	X =  157.000  mm,	Y =  130.000  mm,	Z =   -1.000 mm,
	W =-180.000 deg,	P =   0.000 deg,	R =    90.000 deg
};
P[6603]{
   GP1:
	UF : 1, UT : 3,		CONFIG : 'N U T, 0, 0, 0',
	X =  157.000  mm,	Y =  130.000  mm,	Z =   15.000 mm,
	W =-180.000 deg,	P =   0.000 deg,	R =    90.000 deg
};
P[6745]{
   GP1:
	UF : 1, UT : 3,		CONFIG : 'N U T, 0, 0, 0',
	X =  34.000  mm,	Y =  136.000  mm,	Z =   15.000 mm,
	W =-180.000 deg,	P =   0.000 deg,	R =    90.000 deg
};
P[6746]{
   GP1:
	UF : 1, UT : 3,		CONFIG : 'N U T, 0, 0, 0',
	X =  34.000  mm,	Y =  136.000  mm,	Z =   -1.000 mm,
	W =-180.000 deg,	P =   0.000 deg,	R =    90.000 deg
};
P[6747]{
   GP1:
	UF : 1, UT : 3,		CONFIG : 'N U T, 0, 0, 0',
	X =  34.000  mm,	Y =  136.000  mm,	Z =   15.000 mm,
	W =-180.000 deg,	P =   0.000 deg,	R =    90.000 deg
};
P[6778]{
   GP1:
	UF : 1, UT : 3,		CONFIG : 'N U T, 0, 0, 0',
	X =  106.000  mm,	Y =  136.000  mm,	Z =   15.000 mm,
	W =-180.000 deg,	P =   0.000 deg,	R =    90.000 deg
};
P[6779]{
   GP1:
	UF : 1, UT : 3,		CONFIG : 'N U T, 0, 0, 0',
	X =  106.000  mm,	Y =  136.000  mm,	Z =   -1.000 mm,
	W =-180.000 deg,	P =   0.000 deg,	R =    90.000 deg
};
P[6780]{
   GP1:
	UF : 1, UT : 3,		CONFIG : 'N U T, 0, 0, 0',
	X =  106.000  mm,	Y =  136.000  mm,	Z =   15.000 mm,
	W =-180.000 deg,	P =   0.000 deg,	R =    90.000 deg
};
P[6988]{
   GP1:
	UF : 1, UT : 3,		CONFIG : 'N U T, 0, 0, 0',
	X =  94.000  mm,	Y =  142.000  mm,	Z =   15.000 mm,
	W =-180.000 deg,	P =   0.000 deg,	R =    90.000 deg
};
P[6989]{
   GP1:
	UF : 1, UT : 3,		CONFIG : 'N U T, 0, 0, 0',
	X =  94.000  mm,	Y =  142.000  mm,	Z =   -1.000 mm,
	W =-180.000 deg,	P =   0.000 deg,	R =    90.000 deg
};
P[6990]{
   GP1:
	UF : 1, UT : 3,		CONFIG : 'N U T, 0, 0, 0',
	X =  94.000  mm,	Y =  142.000  mm,	Z =   15.000 mm,
	W =-180.000 deg,	P =   0.000 deg,	R =    90.000 deg
};
P[7054]{
   GP1:
	UF : 1, UT : 3,		CONFIG : 'N U T, 0, 0, 0',
	X =  22.000  mm,	Y =  145.000  mm,	Z =   15.000 mm,
	W =-180.000 deg,	P =   0.000 deg,	R =    90.000 deg
};
P[7055]{
   GP1:
	UF : 1, UT : 3,		CONFIG : 'N U T, 0, 0, 0',
	X =  22.000  mm,	Y =  145.000  mm,	Z =   -1.000 mm,
	W =-180.000 deg,	P =   0.000 deg,	R =    90.000 deg
};
P[7056]{
   GP1:
	UF : 1, UT : 3,		CONFIG : 'N U T, 0, 0, 0',
	X =  22.000  mm,	Y =  145.000  mm,	Z =   15.000 mm,
	W =-180.000 deg,	P =   0.000 deg,	R =    90.000 deg
};
P[7312]{
   GP1:
	UF : 1, UT : 3,		CONFIG : 'N U T, 0, 0, 0',
	X =  109.000  mm,	Y =  151.000  mm,	Z =   15.000 mm,
	W =-180.000 deg,	P =   0.000 deg,	R =    90.000 deg
};
P[7313]{
   GP1:
	UF : 1, UT : 3,		CONFIG : 'N U T, 0, 0, 0',
	X =  109.000  mm,	Y =  151.000  mm,	Z =   -1.000 mm,
	W =-180.000 deg,	P =   0.000 deg,	R =    90.000 deg
};
P[7314]{
   GP1:
	UF : 1, UT : 3,		CONFIG : 'N U T, 0, 0, 0',
	X =  109.000  mm,	Y =  151.000  mm,	Z =   15.000 mm,
	W =-180.000 deg,	P =   0.000 deg,	R =    90.000 deg
};
P[7414]{
   GP1:
	UF : 1, UT : 3,		CONFIG : 'N U T, 0, 0, 0',
	X =  67.000  mm,	Y =  154.000  mm,	Z =   15.000 mm,
	W =-180.000 deg,	P =   0.000 deg,	R =    90.000 deg
};
P[7415]{
   GP1:
	UF : 1, UT : 3,		CONFIG : 'N U T, 0, 0, 0',
	X =  67.000  mm,	Y =  154.000  mm,	Z =   -1.000 mm,
	W =-180.000 deg,	P =   0.000 deg,	R =    90.000 deg
};
P[7416]{
   GP1:
	UF : 1, UT : 3,		CONFIG : 'N U T, 0, 0, 0',
	X =  67.000  mm,	Y =  154.000  mm,	Z =   15.000 mm,
	W =-180.000 deg,	P =   0.000 deg,	R =    90.000 deg
};
P[7657]{
   GP1:
	UF : 1, UT : 3,		CONFIG : 'N U T, 0, 0, 0',
	X =  151.000  mm,	Y =  160.000  mm,	Z =   15.000 mm,
	W =-180.000 deg,	P =   0.000 deg,	R =    90.000 deg
};
P[7658]{
   GP1:
	UF : 1, UT : 3,		CONFIG : 'N U T, 0, 0, 0',
	X =  151.000  mm,	Y =  160.000  mm,	Z =   -1.000 mm,
	W =-180.000 deg,	P =   0.000 deg,	R =    90.000 deg
};
P[7659]{
   GP1:
	UF : 1, UT : 3,		CONFIG : 'N U T, 0, 0, 0',
	X =  151.000  mm,	Y =  160.000  mm,	Z =   15.000 mm,
	W =-180.000 deg,	P =   0.000 deg,	R =    90.000 deg
};
P[7660]{
   GP1:
	UF : 1, UT : 3,		CONFIG : 'N U T, 0, 0, 0',
	X =  154.000  mm,	Y =  160.000  mm,	Z =   15.000 mm,
	W =-180.000 deg,	P =   0.000 deg,	R =    90.000 deg
};
P[7661]{
   GP1:
	UF : 1, UT : 3,		CONFIG : 'N U T, 0, 0, 0',
	X =  154.000  mm,	Y =  160.000  mm,	Z =   -1.000 mm,
	W =-180.000 deg,	P =   0.000 deg,	R =    90.000 deg
};
P[7662]{
   GP1:
	UF : 1, UT : 3,		CONFIG : 'N U T, 0, 0, 0',
	X =  154.000  mm,	Y =  160.000  mm,	Z =   15.000 mm,
	W =-180.000 deg,	P =   0.000 deg,	R =    90.000 deg
};
P[7699]{
   GP1:
	UF : 1, UT : 3,		CONFIG : 'N U T, 0, 0, 0',
	X =  58.000  mm,	Y =  163.000  mm,	Z =   15.000 mm,
	W =-180.000 deg,	P =   0.000 deg,	R =    90.000 deg
};
P[7700]{
   GP1:
	UF : 1, UT : 3,		CONFIG : 'N U T, 0, 0, 0',
	X =  58.000  mm,	Y =  163.000  mm,	Z =   -1.000 mm,
	W =-180.000 deg,	P =   0.000 deg,	R =    90.000 deg
};
P[7701]{
   GP1:
	UF : 1, UT : 3,		CONFIG : 'N U T, 0, 0, 0',
	X =  58.000  mm,	Y =  163.000  mm,	Z =   15.000 mm,
	W =-180.000 deg,	P =   0.000 deg,	R =    90.000 deg
};
P[7705]{
   GP1:
	UF : 1, UT : 3,		CONFIG : 'N U T, 0, 0, 0',
	X =  106.000  mm,	Y =  163.000  mm,	Z =   15.000 mm,
	W =-180.000 deg,	P =   0.000 deg,	R =    90.000 deg
};
P[7706]{
   GP1:
	UF : 1, UT : 3,		CONFIG : 'N U T, 0, 0, 0',
	X =  106.000  mm,	Y =  163.000  mm,	Z =   -1.000 mm,
	W =-180.000 deg,	P =   0.000 deg,	R =    90.000 deg
};
P[7707]{
   GP1:
	UF : 1, UT : 3,		CONFIG : 'N U T, 0, 0, 0',
	X =  106.000  mm,	Y =  163.000  mm,	Z =   15.000 mm,
	W =-180.000 deg,	P =   0.000 deg,	R =    90.000 deg
};
P[7750]{
   GP1:
	UF : 1, UT : 3,		CONFIG : 'N U T, 0, 0, 0',
	X =  151.000  mm,	Y =  163.000  mm,	Z =   15.000 mm,
	W =-180.000 deg,	P =   0.000 deg,	R =    90.000 deg
};
P[7751]{
   GP1:
	UF : 1, UT : 3,		CONFIG : 'N U T, 0, 0, 0',
	X =  151.000  mm,	Y =  163.000  mm,	Z =   -1.000 mm,
	W =-180.000 deg,	P =   0.000 deg,	R =    90.000 deg
};
P[7752]{
   GP1:
	UF : 1, UT : 3,		CONFIG : 'N U T, 0, 0, 0',
	X =  151.000  mm,	Y =  163.000  mm,	Z =   15.000 mm,
	W =-180.000 deg,	P =   0.000 deg,	R =    90.000 deg
};
P[7753]{
   GP1:
	UF : 1, UT : 3,		CONFIG : 'N U T, 0, 0, 0',
	X =  154.000  mm,	Y =  163.000  mm,	Z =   15.000 mm,
	W =-180.000 deg,	P =   0.000 deg,	R =    90.000 deg
};
P[7754]{
   GP1:
	UF : 1, UT : 3,		CONFIG : 'N U T, 0, 0, 0',
	X =  154.000  mm,	Y =  163.000  mm,	Z =   -1.000 mm,
	W =-180.000 deg,	P =   0.000 deg,	R =    90.000 deg
};
P[7755]{
   GP1:
	UF : 1, UT : 3,		CONFIG : 'N U T, 0, 0, 0',
	X =  154.000  mm,	Y =  163.000  mm,	Z =   15.000 mm,
	W =-180.000 deg,	P =   0.000 deg,	R =    90.000 deg
};
P[7792]{
   GP1:
	UF : 1, UT : 3,		CONFIG : 'N U T, 0, 0, 0',
	X =  106.000  mm,	Y =  166.000  mm,	Z =   15.000 mm,
	W =-180.000 deg,	P =   0.000 deg,	R =    90.000 deg
};
P[7793]{
   GP1:
	UF : 1, UT : 3,		CONFIG : 'N U T, 0, 0, 0',
	X =  106.000  mm,	Y =  166.000  mm,	Z =   -1.000 mm,
	W =-180.000 deg,	P =   0.000 deg,	R =    90.000 deg
};
P[7794]{
   GP1:
	UF : 1, UT : 3,		CONFIG : 'N U T, 0, 0, 0',
	X =  106.000  mm,	Y =  166.000  mm,	Z =   15.000 mm,
	W =-180.000 deg,	P =   0.000 deg,	R =    90.000 deg
};
P[7843]{
   GP1:
	UF : 1, UT : 3,		CONFIG : 'N U T, 0, 0, 0',
	X =  28.000  mm,	Y =  169.000  mm,	Z =   15.000 mm,
	W =-180.000 deg,	P =   0.000 deg,	R =    90.000 deg
};
P[7844]{
   GP1:
	UF : 1, UT : 3,		CONFIG : 'N U T, 0, 0, 0',
	X =  28.000  mm,	Y =  169.000  mm,	Z =   -1.000 mm,
	W =-180.000 deg,	P =   0.000 deg,	R =    90.000 deg
};
P[7845]{
   GP1:
	UF : 1, UT : 3,		CONFIG : 'N U T, 0, 0, 0',
	X =  28.000  mm,	Y =  169.000  mm,	Z =   15.000 mm,
	W =-180.000 deg,	P =   0.000 deg,	R =    90.000 deg
};
P[7852]{
   GP1:
	UF : 1, UT : 3,		CONFIG : 'N U T, 0, 0, 0',
	X =  37.000  mm,	Y =  169.000  mm,	Z =   15.000 mm,
	W =-180.000 deg,	P =   0.000 deg,	R =    90.000 deg
};
P[7853]{
   GP1:
	UF : 1, UT : 3,		CONFIG : 'N U T, 0, 0, 0',
	X =  37.000  mm,	Y =  169.000  mm,	Z =   -1.000 mm,
	W =-180.000 deg,	P =   0.000 deg,	R =    90.000 deg
};
P[7854]{
   GP1:
	UF : 1, UT : 3,		CONFIG : 'N U T, 0, 0, 0',
	X =  37.000  mm,	Y =  169.000  mm,	Z =   15.000 mm,
	W =-180.000 deg,	P =   0.000 deg,	R =    90.000 deg
};
P[7858]{
   GP1:
	UF : 1, UT : 3,		CONFIG : 'N U T, 0, 0, 0',
	X =  43.000  mm,	Y =  169.000  mm,	Z =   15.000 mm,
	W =-180.000 deg,	P =   0.000 deg,	R =    90.000 deg
};
P[7859]{
   GP1:
	UF : 1, UT : 3,		CONFIG : 'N U T, 0, 0, 0',
	X =  43.000  mm,	Y =  169.000  mm,	Z =   -1.000 mm,
	W =-180.000 deg,	P =   0.000 deg,	R =    90.000 deg
};
P[7860]{
   GP1:
	UF : 1, UT : 3,		CONFIG : 'N U T, 0, 0, 0',
	X =  43.000  mm,	Y =  169.000  mm,	Z =   15.000 mm,
	W =-180.000 deg,	P =   0.000 deg,	R =    90.000 deg
};
P[7927]{
   GP1:
	UF : 1, UT : 3,		CONFIG : 'N U T, 0, 0, 0',
	X =  34.000  mm,	Y =  172.000  mm,	Z =   15.000 mm,
	W =-180.000 deg,	P =   0.000 deg,	R =    90.000 deg
};
P[7928]{
   GP1:
	UF : 1, UT : 3,		CONFIG : 'N U T, 0, 0, 0',
	X =  34.000  mm,	Y =  172.000  mm,	Z =   -1.000 mm,
	W =-180.000 deg,	P =   0.000 deg,	R =    90.000 deg
};
P[7929]{
   GP1:
	UF : 1, UT : 3,		CONFIG : 'N U T, 0, 0, 0',
	X =  34.000  mm,	Y =  172.000  mm,	Z =   15.000 mm,
	W =-180.000 deg,	P =   0.000 deg,	R =    90.000 deg
};
P[7930]{
   GP1:
	UF : 1, UT : 3,		CONFIG : 'N U T, 0, 0, 0',
	X =  40.000  mm,	Y =  172.000  mm,	Z =   15.000 mm,
	W =-180.000 deg,	P =   0.000 deg,	R =    90.000 deg
};
P[7931]{
   GP1:
	UF : 1, UT : 3,		CONFIG : 'N U T, 0, 0, 0',
	X =  40.000  mm,	Y =  172.000  mm,	Z =   -1.000 mm,
	W =-180.000 deg,	P =   0.000 deg,	R =    90.000 deg
};
P[7932]{
   GP1:
	UF : 1, UT : 3,		CONFIG : 'N U T, 0, 0, 0',
	X =  40.000  mm,	Y =  172.000  mm,	Z =   15.000 mm,
	W =-180.000 deg,	P =   0.000 deg,	R =    90.000 deg
};
P[7936]{
   GP1:
	UF : 1, UT : 3,		CONFIG : 'N U T, 0, 0, 0',
	X =  46.000  mm,	Y =  172.000  mm,	Z =   15.000 mm,
	W =-180.000 deg,	P =   0.000 deg,	R =    90.000 deg
};
P[7937]{
   GP1:
	UF : 1, UT : 3,		CONFIG : 'N U T, 0, 0, 0',
	X =  46.000  mm,	Y =  172.000  mm,	Z =   -1.000 mm,
	W =-180.000 deg,	P =   0.000 deg,	R =    90.000 deg
};
P[7938]{
   GP1:
	UF : 1, UT : 3,		CONFIG : 'N U T, 0, 0, 0',
	X =  46.000  mm,	Y =  172.000  mm,	Z =   15.000 mm,
	W =-180.000 deg,	P =   0.000 deg,	R =    90.000 deg
};
P[7987]{
   GP1:
	UF : 1, UT : 3,		CONFIG : 'N U T, 0, 0, 0',
	X =  148.000  mm,	Y =  172.000  mm,	Z =   15.000 mm,
	W =-180.000 deg,	P =   0.000 deg,	R =    90.000 deg
};
P[7988]{
   GP1:
	UF : 1, UT : 3,		CONFIG : 'N U T, 0, 0, 0',
	X =  148.000  mm,	Y =  172.000  mm,	Z =   -1.000 mm,
	W =-180.000 deg,	P =   0.000 deg,	R =    90.000 deg
};
P[7989]{
   GP1:
	UF : 1, UT : 3,		CONFIG : 'N U T, 0, 0, 0',
	X =  148.000  mm,	Y =  172.000  mm,	Z =   15.000 mm,
	W =-180.000 deg,	P =   0.000 deg,	R =    90.000 deg
};
P[8002]{
   GP1:
	UF : 1, UT : 3,		CONFIG : 'N U T, 0, 0, 0',
	X =  43.000  mm,	Y =  175.000  mm,	Z =   15.000 mm,
	W =-180.000 deg,	P =   0.000 deg,	R =    90.000 deg
};
P[8003]{
   GP1:
	UF : 1, UT : 3,		CONFIG : 'N U T, 0, 0, 0',
	X =  43.000  mm,	Y =  175.000  mm,	Z =   -1.000 mm,
	W =-180.000 deg,	P =   0.000 deg,	R =    90.000 deg
};
P[8004]{
   GP1:
	UF : 1, UT : 3,		CONFIG : 'N U T, 0, 0, 0',
	X =  43.000  mm,	Y =  175.000  mm,	Z =   15.000 mm,
	W =-180.000 deg,	P =   0.000 deg,	R =    90.000 deg
};
P[8005]{
   GP1:
	UF : 1, UT : 3,		CONFIG : 'N U T, 0, 0, 0',
	X =  46.000  mm,	Y =  175.000  mm,	Z =   15.000 mm,
	W =-180.000 deg,	P =   0.000 deg,	R =    90.000 deg
};
P[8006]{
   GP1:
	UF : 1, UT : 3,		CONFIG : 'N U T, 0, 0, 0',
	X =  46.000  mm,	Y =  175.000  mm,	Z =   -1.000 mm,
	W =-180.000 deg,	P =   0.000 deg,	R =    90.000 deg
};
P[8007]{
   GP1:
	UF : 1, UT : 3,		CONFIG : 'N U T, 0, 0, 0',
	X =  46.000  mm,	Y =  175.000  mm,	Z =   15.000 mm,
	W =-180.000 deg,	P =   0.000 deg,	R =    90.000 deg
};
P[8011]{
   GP1:
	UF : 1, UT : 3,		CONFIG : 'N U T, 0, 0, 0',
	X =  109.000  mm,	Y =  175.000  mm,	Z =   15.000 mm,
	W =-180.000 deg,	P =   0.000 deg,	R =    90.000 deg
};
P[8012]{
   GP1:
	UF : 1, UT : 3,		CONFIG : 'N U T, 0, 0, 0',
	X =  109.000  mm,	Y =  175.000  mm,	Z =   -1.000 mm,
	W =-180.000 deg,	P =   0.000 deg,	R =    90.000 deg
};
P[8013]{
   GP1:
	UF : 1, UT : 3,		CONFIG : 'N U T, 0, 0, 0',
	X =  109.000  mm,	Y =  175.000  mm,	Z =   15.000 mm,
	W =-180.000 deg,	P =   0.000 deg,	R =    90.000 deg
};
P[8047]{
   GP1:
	UF : 1, UT : 3,		CONFIG : 'N U T, 0, 0, 0',
	X =  145.000  mm,	Y =  175.000  mm,	Z =   15.000 mm,
	W =-180.000 deg,	P =   0.000 deg,	R =    90.000 deg
};
P[8048]{
   GP1:
	UF : 1, UT : 3,		CONFIG : 'N U T, 0, 0, 0',
	X =  145.000  mm,	Y =  175.000  mm,	Z =   -1.000 mm,
	W =-180.000 deg,	P =   0.000 deg,	R =    90.000 deg
};
P[8049]{
   GP1:
	UF : 1, UT : 3,		CONFIG : 'N U T, 0, 0, 0',
	X =  145.000  mm,	Y =  175.000  mm,	Z =   15.000 mm,
	W =-180.000 deg,	P =   0.000 deg,	R =    90.000 deg
};
P[8077]{
   GP1:
	UF : 1, UT : 3,		CONFIG : 'N U T, 0, 0, 0',
	X =  112.000  mm,	Y =  178.000  mm,	Z =   15.000 mm,
	W =-180.000 deg,	P =   0.000 deg,	R =    90.000 deg
};
P[8078]{
   GP1:
	UF : 1, UT : 3,		CONFIG : 'N U T, 0, 0, 0',
	X =  112.000  mm,	Y =  178.000  mm,	Z =   -1.000 mm,
	W =-180.000 deg,	P =   0.000 deg,	R =    90.000 deg
};
P[8079]{
   GP1:
	UF : 1, UT : 3,		CONFIG : 'N U T, 0, 0, 0',
	X =  112.000  mm,	Y =  178.000  mm,	Z =   15.000 mm,
	W =-180.000 deg,	P =   0.000 deg,	R =    90.000 deg
};
P[8161]{
   GP1:
	UF : 1, UT : 3,		CONFIG : 'N U T, 0, 0, 0',
	X =  112.000  mm,	Y =  181.000  mm,	Z =   15.000 mm,
	W =-180.000 deg,	P =   0.000 deg,	R =    90.000 deg
};
P[8162]{
   GP1:
	UF : 1, UT : 3,		CONFIG : 'N U T, 0, 0, 0',
	X =  112.000  mm,	Y =  181.000  mm,	Z =   -1.000 mm,
	W =-180.000 deg,	P =   0.000 deg,	R =    90.000 deg
};
P[8163]{
   GP1:
	UF : 1, UT : 3,		CONFIG : 'N U T, 0, 0, 0',
	X =  112.000  mm,	Y =  181.000  mm,	Z =   15.000 mm,
	W =-180.000 deg,	P =   0.000 deg,	R =    90.000 deg
};
P[8197]{
   GP1:
	UF : 1, UT : 3,		CONFIG : 'N U T, 0, 0, 0',
	X =  148.000  mm,	Y =  181.000  mm,	Z =   15.000 mm,
	W =-180.000 deg,	P =   0.000 deg,	R =    90.000 deg
};
P[8198]{
   GP1:
	UF : 1, UT : 3,		CONFIG : 'N U T, 0, 0, 0',
	X =  148.000  mm,	Y =  181.000  mm,	Z =   -1.000 mm,
	W =-180.000 deg,	P =   0.000 deg,	R =    90.000 deg
};
P[8199]{
   GP1:
	UF : 1, UT : 3,		CONFIG : 'N U T, 0, 0, 0',
	X =  148.000  mm,	Y =  181.000  mm,	Z =   15.000 mm,
	W =-180.000 deg,	P =   0.000 deg,	R =    90.000 deg
};
P[8275]{
   GP1:
	UF : 1, UT : 3,		CONFIG : 'N U T, 0, 0, 0',
	X =  124.000  mm,	Y =  184.000  mm,	Z =   15.000 mm,
	W =-180.000 deg,	P =   0.000 deg,	R =    90.000 deg
};
P[8276]{
   GP1:
	UF : 1, UT : 3,		CONFIG : 'N U T, 0, 0, 0',
	X =  124.000  mm,	Y =  184.000  mm,	Z =   -1.000 mm,
	W =-180.000 deg,	P =   0.000 deg,	R =    90.000 deg
};
P[8277]{
   GP1:
	UF : 1, UT : 3,		CONFIG : 'N U T, 0, 0, 0',
	X =  124.000  mm,	Y =  184.000  mm,	Z =   15.000 mm,
	W =-180.000 deg,	P =   0.000 deg,	R =    90.000 deg
};
P[8281]{
   GP1:
	UF : 1, UT : 3,		CONFIG : 'N U T, 0, 0, 0',
	X =  130.000  mm,	Y =  184.000  mm,	Z =   15.000 mm,
	W =-180.000 deg,	P =   0.000 deg,	R =    90.000 deg
};
P[8282]{
   GP1:
	UF : 1, UT : 3,		CONFIG : 'N U T, 0, 0, 0',
	X =  130.000  mm,	Y =  184.000  mm,	Z =   -1.000 mm,
	W =-180.000 deg,	P =   0.000 deg,	R =    90.000 deg
};
P[8283]{
   GP1:
	UF : 1, UT : 3,		CONFIG : 'N U T, 0, 0, 0',
	X =  130.000  mm,	Y =  184.000  mm,	Z =   15.000 mm,
	W =-180.000 deg,	P =   0.000 deg,	R =    90.000 deg
};
P[8284]{
   GP1:
	UF : 1, UT : 3,		CONFIG : 'N U T, 0, 0, 0',
	X =  133.000  mm,	Y =  184.000  mm,	Z =   15.000 mm,
	W =-180.000 deg,	P =   0.000 deg,	R =    90.000 deg
};
P[8285]{
   GP1:
	UF : 1, UT : 3,		CONFIG : 'N U T, 0, 0, 0',
	X =  133.000  mm,	Y =  184.000  mm,	Z =   -1.000 mm,
	W =-180.000 deg,	P =   0.000 deg,	R =    90.000 deg
};
P[8286]{
   GP1:
	UF : 1, UT : 3,		CONFIG : 'N U T, 0, 0, 0',
	X =  133.000  mm,	Y =  184.000  mm,	Z =   15.000 mm,
	W =-180.000 deg,	P =   0.000 deg,	R =    90.000 deg
};
P[8287]{
   GP1:
	UF : 1, UT : 3,		CONFIG : 'N U T, 0, 0, 0',
	X =  136.000  mm,	Y =  184.000  mm,	Z =   15.000 mm,
	W =-180.000 deg,	P =   0.000 deg,	R =    90.000 deg
};
P[8288]{
   GP1:
	UF : 1, UT : 3,		CONFIG : 'N U T, 0, 0, 0',
	X =  136.000  mm,	Y =  184.000  mm,	Z =   -1.000 mm,
	W =-180.000 deg,	P =   0.000 deg,	R =    90.000 deg
};
P[8289]{
   GP1:
	UF : 1, UT : 3,		CONFIG : 'N U T, 0, 0, 0',
	X =  136.000  mm,	Y =  184.000  mm,	Z =   15.000 mm,
	W =-180.000 deg,	P =   0.000 deg,	R =    90.000 deg
};
P[8398]{
   GP1:
	UF : 1, UT : 3,		CONFIG : 'N U T, 0, 0, 0',
	X =  70.000  mm,	Y =  187.000  mm,	Z =   15.000 mm,
	W =-180.000 deg,	P =   0.000 deg,	R =    90.000 deg
};
P[8399]{
   GP1:
	UF : 1, UT : 3,		CONFIG : 'N U T, 0, 0, 0',
	X =  70.000  mm,	Y =  187.000  mm,	Z =   -1.000 mm,
	W =-180.000 deg,	P =   0.000 deg,	R =    90.000 deg
};
P[8400]{
   GP1:
	UF : 1, UT : 3,		CONFIG : 'N U T, 0, 0, 0',
	X =  70.000  mm,	Y =  187.000  mm,	Z =   15.000 mm,
	W =-180.000 deg,	P =   0.000 deg,	R =    90.000 deg
};
P[8452]{
   GP1:
	UF : 1, UT : 3,		CONFIG : 'N U T, 0, 0, 0',
	X =  124.000  mm,	Y =  187.000  mm,	Z =   15.000 mm,
	W =-180.000 deg,	P =   0.000 deg,	R =    90.000 deg
};
P[8453]{
   GP1:
	UF : 1, UT : 3,		CONFIG : 'N U T, 0, 0, 0',
	X =  124.000  mm,	Y =  187.000  mm,	Z =   -1.000 mm,
	W =-180.000 deg,	P =   0.000 deg,	R =    90.000 deg
};
P[8454]{
   GP1:
	UF : 1, UT : 3,		CONFIG : 'N U T, 0, 0, 0',
	X =  124.000  mm,	Y =  187.000  mm,	Z =   15.000 mm,
	W =-180.000 deg,	P =   0.000 deg,	R =    90.000 deg
};
P[8455]{
   GP1:
	UF : 1, UT : 3,		CONFIG : 'N U T, 0, 0, 0',
	X =  127.000  mm,	Y =  187.000  mm,	Z =   15.000 mm,
	W =-180.000 deg,	P =   0.000 deg,	R =    90.000 deg
};
P[8456]{
   GP1:
	UF : 1, UT : 3,		CONFIG : 'N U T, 0, 0, 0',
	X =  127.000  mm,	Y =  187.000  mm,	Z =   -1.000 mm,
	W =-180.000 deg,	P =   0.000 deg,	R =    90.000 deg
};
P[8457]{
   GP1:
	UF : 1, UT : 3,		CONFIG : 'N U T, 0, 0, 0',
	X =  127.000  mm,	Y =  187.000  mm,	Z =   15.000 mm,
	W =-180.000 deg,	P =   0.000 deg,	R =    90.000 deg
};
P[8461]{
   GP1:
	UF : 1, UT : 3,		CONFIG : 'N U T, 0, 0, 0',
	X =  133.000  mm,	Y =  187.000  mm,	Z =   15.000 mm,
	W =-180.000 deg,	P =   0.000 deg,	R =    90.000 deg
};
P[8462]{
   GP1:
	UF : 1, UT : 3,		CONFIG : 'N U T, 0, 0, 0',
	X =  133.000  mm,	Y =  187.000  mm,	Z =   -1.000 mm,
	W =-180.000 deg,	P =   0.000 deg,	R =    90.000 deg
};
P[8463]{
   GP1:
	UF : 1, UT : 3,		CONFIG : 'N U T, 0, 0, 0',
	X =  133.000  mm,	Y =  187.000  mm,	Z =   15.000 mm,
	W =-180.000 deg,	P =   0.000 deg,	R =    90.000 deg
};
P[8464]{
   GP1:
	UF : 1, UT : 3,		CONFIG : 'N U T, 0, 0, 0',
	X =  136.000  mm,	Y =  187.000  mm,	Z =   15.000 mm,
	W =-180.000 deg,	P =   0.000 deg,	R =    90.000 deg
};
P[8465]{
   GP1:
	UF : 1, UT : 3,		CONFIG : 'N U T, 0, 0, 0',
	X =  136.000  mm,	Y =  187.000  mm,	Z =   -1.000 mm,
	W =-180.000 deg,	P =   0.000 deg,	R =    90.000 deg
};
P[8466]{
   GP1:
	UF : 1, UT : 3,		CONFIG : 'N U T, 0, 0, 0',
	X =  136.000  mm,	Y =  187.000  mm,	Z =   15.000 mm,
	W =-180.000 deg,	P =   0.000 deg,	R =    90.000 deg
};
P[11569]{
   GP1:
	UF : 1, UT : 3,		CONFIG : 'N U T, 0, 0, 0',
	X =  145.000  mm,	Y =  300.000  mm,	Z =   100.000 mm,
	W =-180.000 deg,	P =   0.000 deg,	R =    90.000 deg
};
/END
